// TIA Portal V20 export
FUNCTION_BLOCK "Sequence_1_SideTapeLoading"   // FB32854, LAD
TITLE = Sequence
// Sequence template programmend in ladder logic
// stored: IsIECCheckEnabled true, MemoryReserve 100, Namespace Unit1.Em4, SetENOAutomatically true
   VAR_INPUT
      unitStatus { ExternalAccessible := 'False'; ExternalVisible := 'False'; ExternalWritable := 'False'} : "LAF_typeUnitStatus";   // Current unit status o be used in this EM
   END_VAR
   VAR
      instSequenceLADControl { ExternalWritable := 'False'} : "LAF_ControlLadSequence";
      instSequenceLADStatus { ExternalWritable := 'False'} : "LAF_StatusLadSequence";
      statTonTime { ExternalWritable := 'False'} : Array[0..9999] of TON_TIME;
   END_VAR
   VAR_TEMP
      tempCustomerAction : Bool;   // Placeholder for possible actions
      tempDo_nothing_and_wait_for_init : Bool;   // Placeholder for doing nothing
      tempSafeStateCondition : Bool;   // Temp Condition for the equipment module to be in a safe state
   END_VAR
   VAR CONSTANT
      delayTime : Time := T#1000ms;
      STEP_IDLE : DInt := 1;
      JOB_1_STEP_1 : DInt := 101;
      JOB_1_STEP_10 : DInt := 110;
      JOB_1_STEP_20 : DInt := 120;
      JOB_1_STEP_30 : DInt := 130;
      JOB_1_STEP_40 : DInt := 140;
      JOB_1_STEP_50 : DInt := 150;
      JOB_1_STEP_90 : DInt := 190;
      JOB_2_STEP_1 : DInt := 201;
      JOB_2_STEP_10 : DInt := 210;
      JOB_2_STEP_20 : DInt := 220;
      JOB_2_STEP_30 : DInt := 230;
      JOB_2_STEP_40 : DInt := 240;
      JOB_2_STEP_50 : DInt := 250;
      JOB_2_STEP_60 : DInt := 260;
      JOB_2_STEP_90 : DInt := 290;
      JOB_3_STEP_10 : DInt := 310;
      JOB_3_STEP_20 : DInt := 320;
      JOB_3_STEP_30 : DInt := 330;
      JOB_3_STEP_40 : DInt := 340;
      STEP_IMMEDIATE_STOP : DInt := 9001;   // Step executed when an immediate stop command is triggered for the sequence (i.e. when unit is in state aborting)
      TO_DO_INSERT_ACTIONS_HERE : Bool := TRUE;   // Template : Add actions
      TO_DO_INSERT_CONDITION_FOR_TRANSITION_HERE : Bool := TRUE;   // Template : Add conditions
   END_VAR
   VAR_TEMP   // added for the SCL form of the ladder/FBD networks
      _w1 : Bool;
   END_VAR
BEGIN

REGION Network 1: BLOCK INFO HEADER
   // (company) / (C) Copyright (year)
   // ---------------------------------------------------------------------------------
   // Title:                             (Title of this block)
   // Comment/Function: (that is implemented in the block)
   // Library/Family:           (that the source is dedicated to)
   // Author:                        (department / person in charge / contact)
   // Target System:          (test system with FW version)
   // Engineering:              TIA Portal (SW version)
   // Restrictions:               (OB types, etc.)
   // Requirements:           (hardware, technological package, etc.)
   // ---------------------------------------------------------------------------------
   // Change log table:
   // Version          | Date             | Signature      | Expert in charge  | Changes applied ------------------------|----------------------|-------------------------|--------------------------------|-----------------------
   // 001.000.000 | yyyy-mm-dd | 0x00000000 | (name of expert) | First released version
END_REGION

REGION Network 2: DESCRIPTION
   // This is a template block provided by the Automation Framework. It can be used to create an own project.
   // The Block Info Header is prepared to put in your own data.
   // Description of the block could be added here and the docu created by Code2Docu.
END_REGION

REGION Network 3: *************** CONTROL **********************
END_REGION

REGION Network 4: Sequence Control ("Enter your Sequins number here")
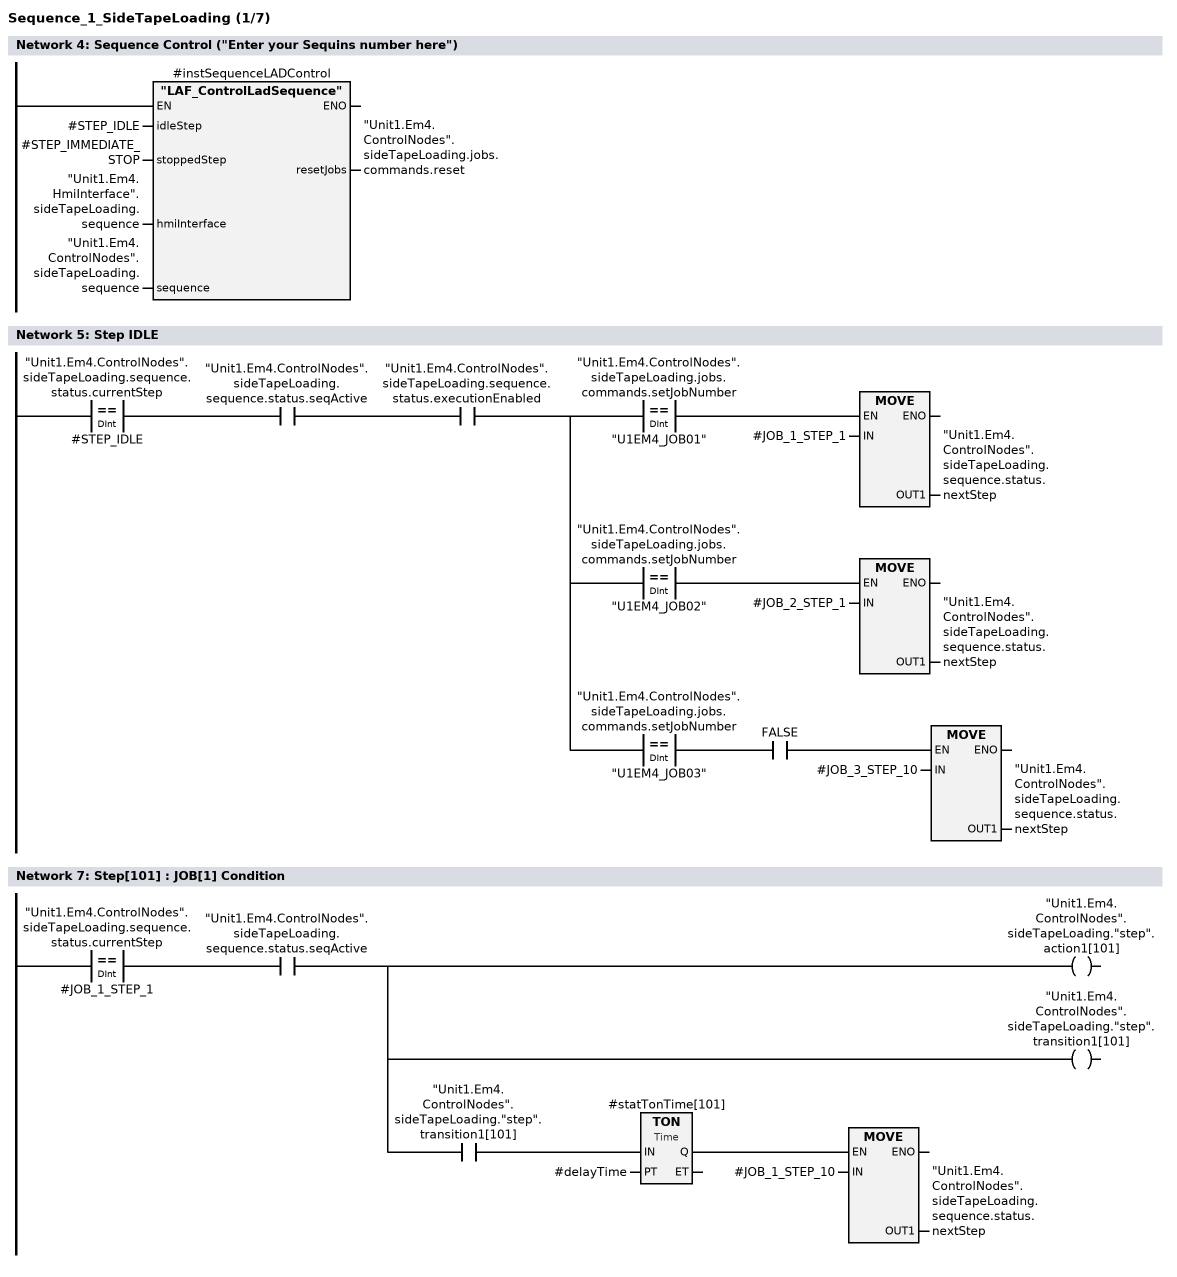
   RUNG wire#powerrail
      #instSequenceLADControl(idleStep := #STEP_IDLE, stoppedStep := #STEP_IMMEDIATE_STOP, hmiInterface := "Unit1.Em4.HmiInterface".sideTapeLoading.sequence, sequence := "Unit1.Em4.ControlNodes".sideTapeLoading.sequence, resetJobs => "Unit1.Em4.ControlNodes".sideTapeLoading.jobs.commands.reset)
   END_RUNG
   // the same network as SCL:
   #instSequenceLADControl(idleStep := #STEP_IDLE,   // "LAF_ControlLadSequence"
                           stoppedStep := #STEP_IMMEDIATE_STOP,
                           hmiInterface := "Unit1.Em4.HmiInterface".sideTapeLoading.sequence,
                           sequence := "Unit1.Em4.ControlNodes".sideTapeLoading.sequence,
                           resetJobs => "Unit1.Em4.ControlNodes".sideTapeLoading.jobs.commands.reset);
END_REGION

REGION Network 5: Step IDLE
   RUNG wire#powerrail
      { S7_Templates := "SrcType := DInt" } EQ_Contact(in1 := "Unit1.Em4.ControlNodes".sideTapeLoading.sequence.status.currentStep, in2 := #STEP_IDLE)
      Contact( "Unit1.Em4.ControlNodes".sideTapeLoading.sequence.status.seqActive )
      Contact( "Unit1.Em4.ControlNodes".sideTapeLoading.sequence.status.executionEnabled )
      wire#w1
      { S7_Templates := "SrcType := DInt" } EQ_Contact(in1 := "Unit1.Em4.ControlNodes".sideTapeLoading.jobs.commands.setJobNumber, in2 := "U1EM4_JOB01")
      Move(in := #JOB_1_STEP_1, out1 => "Unit1.Em4.ControlNodes".sideTapeLoading.sequence.status.nextStep)
   END_RUNG
   RUNG wire#w1
      { S7_Templates := "SrcType := DInt" } EQ_Contact(in1 := "Unit1.Em4.ControlNodes".sideTapeLoading.jobs.commands.setJobNumber, in2 := "U1EM4_JOB02")
      Move(in := #JOB_2_STEP_1, out1 => "Unit1.Em4.ControlNodes".sideTapeLoading.sequence.status.nextStep)
   END_RUNG
   RUNG wire#w1
      { S7_Templates := "SrcType := DInt" } EQ_Contact(in1 := "Unit1.Em4.ControlNodes".sideTapeLoading.jobs.commands.setJobNumber, in2 := "U1EM4_JOB03")
      Contact( FALSE )
      Move(in := #JOB_3_STEP_10, out1 => "Unit1.Em4.ControlNodes".sideTapeLoading.sequence.status.nextStep)
   END_RUNG
   // the same network as SCL:
   #_w1 := ("Unit1.Em4.ControlNodes".sideTapeLoading.sequence.status.currentStep = #STEP_IDLE) AND "Unit1.Em4.ControlNodes".sideTapeLoading.sequence.status.seqActive AND "Unit1.Em4.ControlNodes".sideTapeLoading.sequence.status.executionEnabled;
   IF #_w1 AND ("Unit1.Em4.ControlNodes".sideTapeLoading.jobs.commands.setJobNumber = "U1EM4_JOB01") THEN
       "Unit1.Em4.ControlNodes".sideTapeLoading.sequence.status.nextStep := #JOB_1_STEP_1;
   END_IF;
   IF #_w1 AND ("Unit1.Em4.ControlNodes".sideTapeLoading.jobs.commands.setJobNumber = "U1EM4_JOB02") THEN
       "Unit1.Em4.ControlNodes".sideTapeLoading.sequence.status.nextStep := #JOB_2_STEP_1;
   END_IF;
   IF #_w1 AND ("Unit1.Em4.ControlNodes".sideTapeLoading.jobs.commands.setJobNumber = "U1EM4_JOB03") AND FALSE THEN
       "Unit1.Em4.ControlNodes".sideTapeLoading.sequence.status.nextStep := #JOB_3_STEP_10;
   END_IF;
END_REGION

REGION Network 6: *************** JOB[1] HOMING *************************
END_REGION

REGION Network 7: Step[101] : JOB[1] Condition
   RUNG wire#powerrail
      { S7_Templates := "SrcType := DInt" } EQ_Contact(in1 := "Unit1.Em4.ControlNodes".sideTapeLoading.sequence.status.currentStep, in2 := #JOB_1_STEP_1)
      Contact( "Unit1.Em4.ControlNodes".sideTapeLoading.sequence.status.seqActive )
      wire#w1
      Coil( "Unit1.Em4.ControlNodes".sideTapeLoading."step".action1[101] )
   END_RUNG
   RUNG wire#w1
      Coil( "Unit1.Em4.ControlNodes".sideTapeLoading."step".transition1[101] )
   END_RUNG
   RUNG wire#w1
      Contact( "Unit1.Em4.ControlNodes".sideTapeLoading."step".transition1[101] )
      { S7_Templates := "time_type := Time" } #statTonTime[101].TON(pt := #delayTime, et =>)
      Move(in := #JOB_1_STEP_10, out1 => "Unit1.Em4.ControlNodes".sideTapeLoading.sequence.status.nextStep)
   END_RUNG
   // the same network as SCL:
   "Unit1.Em4.ControlNodes".sideTapeLoading."step".action1[101] := ("Unit1.Em4.ControlNodes".sideTapeLoading.sequence.status.currentStep = #JOB_1_STEP_1) AND "Unit1.Em4.ControlNodes".sideTapeLoading.sequence.status.seqActive;
   "Unit1.Em4.ControlNodes".sideTapeLoading."step".transition1[101] := ("Unit1.Em4.ControlNodes".sideTapeLoading.sequence.status.currentStep = #JOB_1_STEP_1) AND "Unit1.Em4.ControlNodes".sideTapeLoading.sequence.status.seqActive;
   #statTonTime[101].TON(IN := ("Unit1.Em4.ControlNodes".sideTapeLoading.sequence.status.currentStep = #JOB_1_STEP_1) AND "Unit1.Em4.ControlNodes".sideTapeLoading.sequence.status.seqActive AND "Unit1.Em4.ControlNodes".sideTapeLoading."step".transition1[101],
                         PT := #delayTime);
   IF #statTonTime[101].Q THEN
       "Unit1.Em4.ControlNodes".sideTapeLoading.sequence.status.nextStep := #JOB_1_STEP_10;
   END_IF;
END_REGION

REGION Network 8: Step[110] : Side Tape Loading Down
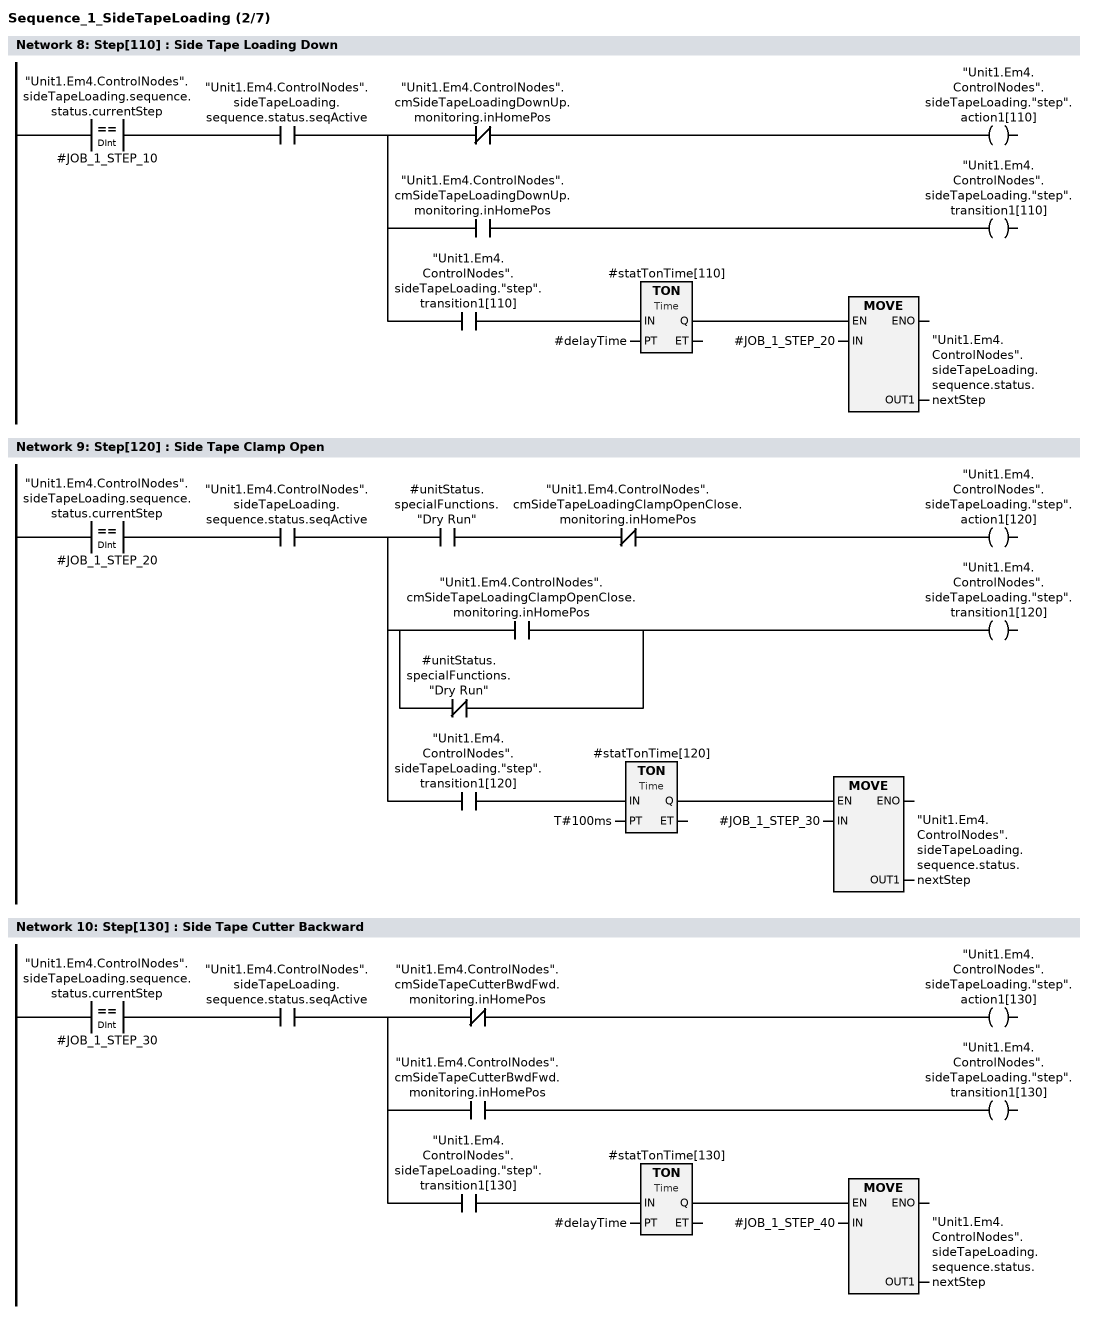
   RUNG wire#powerrail
      { S7_Templates := "SrcType := DInt" } EQ_Contact(in1 := "Unit1.Em4.ControlNodes".sideTapeLoading.sequence.status.currentStep, in2 := #JOB_1_STEP_10)
      Contact( "Unit1.Em4.ControlNodes".sideTapeLoading.sequence.status.seqActive )
      wire#w1
      I_Contact( "Unit1.Em4.ControlNodes".cmSideTapeLoadingDownUp.monitoring.inHomePos )
      Coil( "Unit1.Em4.ControlNodes".sideTapeLoading."step".action1[110] )
   END_RUNG
   RUNG wire#w1
      Contact( "Unit1.Em4.ControlNodes".cmSideTapeLoadingDownUp.monitoring.inHomePos )
      Coil( "Unit1.Em4.ControlNodes".sideTapeLoading."step".transition1[110] )
   END_RUNG
   RUNG wire#w1
      Contact( "Unit1.Em4.ControlNodes".sideTapeLoading."step".transition1[110] )
      { S7_Templates := "time_type := Time" } #statTonTime[110].TON(pt := #delayTime, et =>)
      Move(in := #JOB_1_STEP_20, out1 => "Unit1.Em4.ControlNodes".sideTapeLoading.sequence.status.nextStep)
   END_RUNG
   // the same network as SCL:
   #_w1 := ("Unit1.Em4.ControlNodes".sideTapeLoading.sequence.status.currentStep = #JOB_1_STEP_10) AND "Unit1.Em4.ControlNodes".sideTapeLoading.sequence.status.seqActive;
   "Unit1.Em4.ControlNodes".sideTapeLoading."step".action1[110] := #_w1 AND NOT "Unit1.Em4.ControlNodes".cmSideTapeLoadingDownUp.monitoring.inHomePos;
   "Unit1.Em4.ControlNodes".sideTapeLoading."step".transition1[110] := #_w1 AND "Unit1.Em4.ControlNodes".cmSideTapeLoadingDownUp.monitoring.inHomePos;
   #statTonTime[110].TON(IN := #_w1 AND "Unit1.Em4.ControlNodes".sideTapeLoading."step".transition1[110],
                         PT := #delayTime);
   IF #statTonTime[110].Q THEN
       "Unit1.Em4.ControlNodes".sideTapeLoading.sequence.status.nextStep := #JOB_1_STEP_20;
   END_IF;
END_REGION

REGION Network 9: Step[120] : Side Tape Clamp Open
   RUNG wire#powerrail
      { S7_Templates := "SrcType := DInt" } EQ_Contact(in1 := "Unit1.Em4.ControlNodes".sideTapeLoading.sequence.status.currentStep, in2 := #JOB_1_STEP_20)
      Contact( "Unit1.Em4.ControlNodes".sideTapeLoading.sequence.status.seqActive )
      wire#w1
      Contact( #unitStatus.specialFunctions."Dry Run" )
      I_Contact( "Unit1.Em4.ControlNodes".cmSideTapeLoadingClampOpenClose.monitoring.inHomePos )
      Coil( "Unit1.Em4.ControlNodes".sideTapeLoading."step".action1[120] )
   END_RUNG
   RUNG wire#w1
      Contact( "Unit1.Em4.ControlNodes".cmSideTapeLoadingClampOpenClose.monitoring.inHomePos )
      wire#w2
      Coil( "Unit1.Em4.ControlNodes".sideTapeLoading."step".transition1[120] )
   END_RUNG
   RUNG wire#w1
      I_Contact( #unitStatus.specialFunctions."Dry Run" )
   END_RUNG wire#w2
   RUNG wire#w1
      Contact( "Unit1.Em4.ControlNodes".sideTapeLoading."step".transition1[120] )
      { S7_Templates := "time_type := Time" } #statTonTime[120].TON(pt := T#100ms, et =>)
      Move(in := #JOB_1_STEP_30, out1 => "Unit1.Em4.ControlNodes".sideTapeLoading.sequence.status.nextStep)
   END_RUNG
   // the same network as SCL:
   #_w1 := ("Unit1.Em4.ControlNodes".sideTapeLoading.sequence.status.currentStep = #JOB_1_STEP_20) AND "Unit1.Em4.ControlNodes".sideTapeLoading.sequence.status.seqActive;
   "Unit1.Em4.ControlNodes".sideTapeLoading."step".action1[120] := #_w1 AND #unitStatus.specialFunctions."Dry Run" AND NOT "Unit1.Em4.ControlNodes".cmSideTapeLoadingClampOpenClose.monitoring.inHomePos;
   "Unit1.Em4.ControlNodes".sideTapeLoading."step".transition1[120] := #_w1 AND ("Unit1.Em4.ControlNodes".cmSideTapeLoadingClampOpenClose.monitoring.inHomePos OR NOT #unitStatus.specialFunctions."Dry Run");
   #statTonTime[120].TON(IN := #_w1 AND "Unit1.Em4.ControlNodes".sideTapeLoading."step".transition1[120],
                         PT := T#100ms);
   IF #statTonTime[120].Q THEN
       "Unit1.Em4.ControlNodes".sideTapeLoading.sequence.status.nextStep := #JOB_1_STEP_30;
   END_IF;
END_REGION

REGION Network 10: Step[130] : Side Tape Cutter Backward
   RUNG wire#powerrail
      { S7_Templates := "SrcType := DInt" } EQ_Contact(in1 := "Unit1.Em4.ControlNodes".sideTapeLoading.sequence.status.currentStep, in2 := #JOB_1_STEP_30)
      Contact( "Unit1.Em4.ControlNodes".sideTapeLoading.sequence.status.seqActive )
      wire#w1
      I_Contact( "Unit1.Em4.ControlNodes".cmSideTapeCutterBwdFwd.monitoring.inHomePos )
      Coil( "Unit1.Em4.ControlNodes".sideTapeLoading."step".action1[130] )
   END_RUNG
   RUNG wire#w1
      Contact( "Unit1.Em4.ControlNodes".cmSideTapeCutterBwdFwd.monitoring.inHomePos )
      Coil( "Unit1.Em4.ControlNodes".sideTapeLoading."step".transition1[130] )
   END_RUNG
   RUNG wire#w1
      Contact( "Unit1.Em4.ControlNodes".sideTapeLoading."step".transition1[130] )
      { S7_Templates := "time_type := Time" } #statTonTime[130].TON(pt := #delayTime, et =>)
      Move(in := #JOB_1_STEP_40, out1 => "Unit1.Em4.ControlNodes".sideTapeLoading.sequence.status.nextStep)
   END_RUNG
   // the same network as SCL:
   #_w1 := ("Unit1.Em4.ControlNodes".sideTapeLoading.sequence.status.currentStep = #JOB_1_STEP_30) AND "Unit1.Em4.ControlNodes".sideTapeLoading.sequence.status.seqActive;
   "Unit1.Em4.ControlNodes".sideTapeLoading."step".action1[130] := #_w1 AND NOT "Unit1.Em4.ControlNodes".cmSideTapeCutterBwdFwd.monitoring.inHomePos;
   "Unit1.Em4.ControlNodes".sideTapeLoading."step".transition1[130] := #_w1 AND "Unit1.Em4.ControlNodes".cmSideTapeCutterBwdFwd.monitoring.inHomePos;
   #statTonTime[130].TON(IN := #_w1 AND "Unit1.Em4.ControlNodes".sideTapeLoading."step".transition1[130],
                         PT := #delayTime);
   IF #statTonTime[130].Q THEN
       "Unit1.Em4.ControlNodes".sideTapeLoading.sequence.status.nextStep := #JOB_1_STEP_40;
   END_IF;
END_REGION

REGION Network 11: Step[140] : Side Tape Cutter Clamp Forward
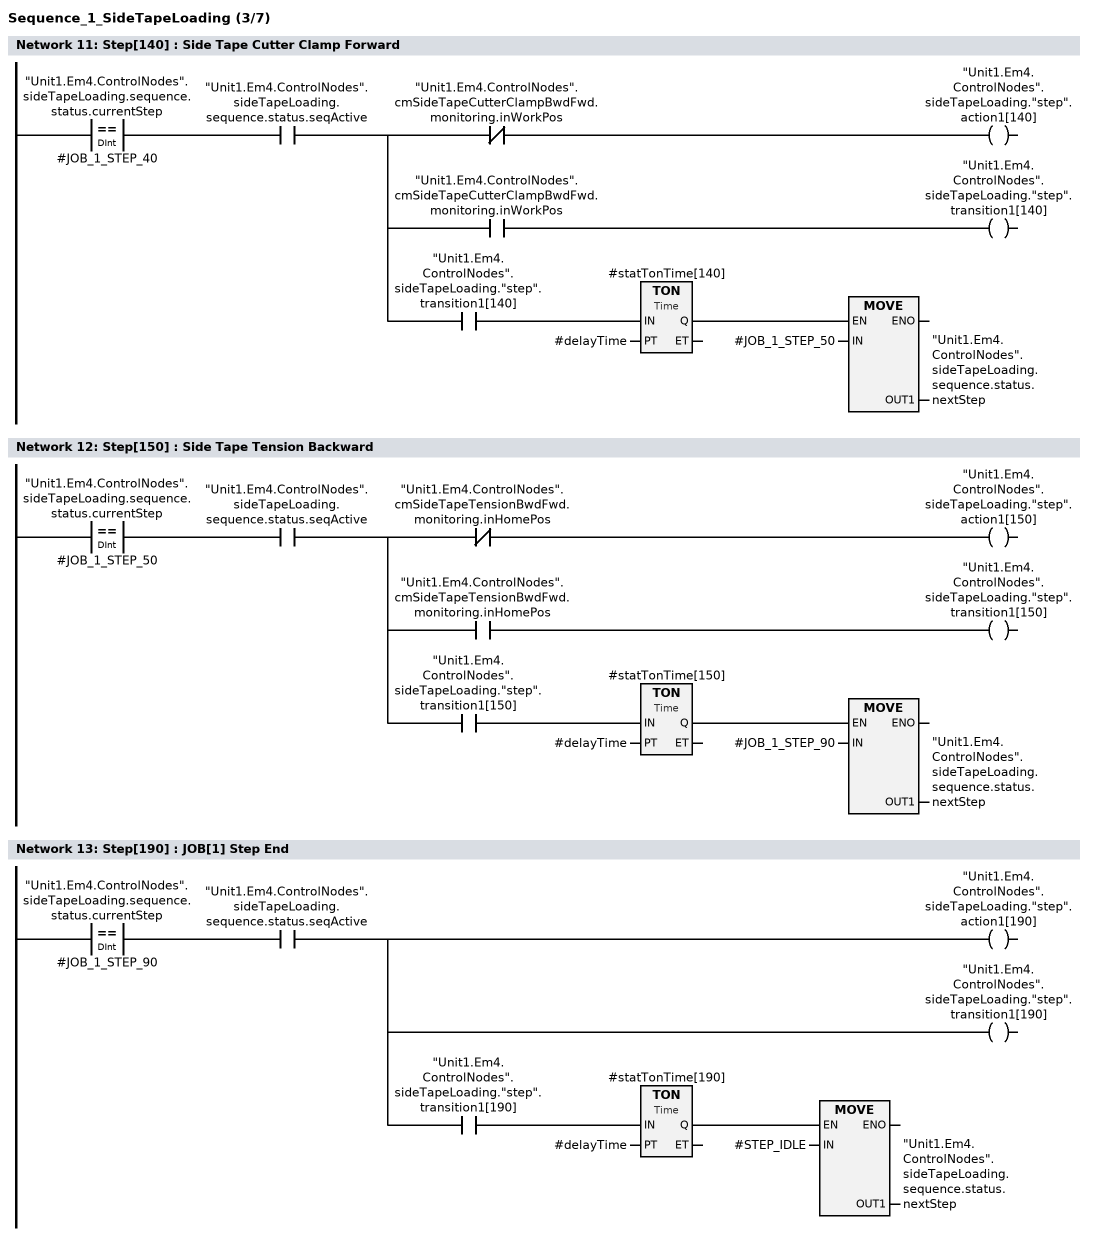
   RUNG wire#powerrail
      { S7_Templates := "SrcType := DInt" } EQ_Contact(in1 := "Unit1.Em4.ControlNodes".sideTapeLoading.sequence.status.currentStep, in2 := #JOB_1_STEP_40)
      Contact( "Unit1.Em4.ControlNodes".sideTapeLoading.sequence.status.seqActive )
      wire#w1
      I_Contact( "Unit1.Em4.ControlNodes".cmSideTapeCutterClampBwdFwd.monitoring.inWorkPos )
      Coil( "Unit1.Em4.ControlNodes".sideTapeLoading."step".action1[140] )
   END_RUNG
   RUNG wire#w1
      Contact( "Unit1.Em4.ControlNodes".cmSideTapeCutterClampBwdFwd.monitoring.inWorkPos )
      Coil( "Unit1.Em4.ControlNodes".sideTapeLoading."step".transition1[140] )
   END_RUNG
   RUNG wire#w1
      Contact( "Unit1.Em4.ControlNodes".sideTapeLoading."step".transition1[140] )
      { S7_Templates := "time_type := Time" } #statTonTime[140].TON(pt := #delayTime, et =>)
      Move(in := #JOB_1_STEP_50, out1 => "Unit1.Em4.ControlNodes".sideTapeLoading.sequence.status.nextStep)
   END_RUNG
   // the same network as SCL:
   #_w1 := ("Unit1.Em4.ControlNodes".sideTapeLoading.sequence.status.currentStep = #JOB_1_STEP_40) AND "Unit1.Em4.ControlNodes".sideTapeLoading.sequence.status.seqActive;
   "Unit1.Em4.ControlNodes".sideTapeLoading."step".action1[140] := #_w1 AND NOT "Unit1.Em4.ControlNodes".cmSideTapeCutterClampBwdFwd.monitoring.inWorkPos;
   "Unit1.Em4.ControlNodes".sideTapeLoading."step".transition1[140] := #_w1 AND "Unit1.Em4.ControlNodes".cmSideTapeCutterClampBwdFwd.monitoring.inWorkPos;
   #statTonTime[140].TON(IN := #_w1 AND "Unit1.Em4.ControlNodes".sideTapeLoading."step".transition1[140],
                         PT := #delayTime);
   IF #statTonTime[140].Q THEN
       "Unit1.Em4.ControlNodes".sideTapeLoading.sequence.status.nextStep := #JOB_1_STEP_50;
   END_IF;
END_REGION

REGION Network 12: Step[150] : Side Tape Tension Backward
   RUNG wire#powerrail
      { S7_Templates := "SrcType := DInt" } EQ_Contact(in1 := "Unit1.Em4.ControlNodes".sideTapeLoading.sequence.status.currentStep, in2 := #JOB_1_STEP_50)
      Contact( "Unit1.Em4.ControlNodes".sideTapeLoading.sequence.status.seqActive )
      wire#w1
      I_Contact( "Unit1.Em4.ControlNodes".cmSideTapeTensionBwdFwd.monitoring.inHomePos )
      Coil( "Unit1.Em4.ControlNodes".sideTapeLoading."step".action1[150] )
   END_RUNG
   RUNG wire#w1
      Contact( "Unit1.Em4.ControlNodes".cmSideTapeTensionBwdFwd.monitoring.inHomePos )
      Coil( "Unit1.Em4.ControlNodes".sideTapeLoading."step".transition1[150] )
   END_RUNG
   RUNG wire#w1
      Contact( "Unit1.Em4.ControlNodes".sideTapeLoading."step".transition1[150] )
      { S7_Templates := "time_type := Time" } #statTonTime[150].TON(pt := #delayTime, et =>)
      Move(in := #JOB_1_STEP_90, out1 => "Unit1.Em4.ControlNodes".sideTapeLoading.sequence.status.nextStep)
   END_RUNG
   // the same network as SCL:
   #_w1 := ("Unit1.Em4.ControlNodes".sideTapeLoading.sequence.status.currentStep = #JOB_1_STEP_50) AND "Unit1.Em4.ControlNodes".sideTapeLoading.sequence.status.seqActive;
   "Unit1.Em4.ControlNodes".sideTapeLoading."step".action1[150] := #_w1 AND NOT "Unit1.Em4.ControlNodes".cmSideTapeTensionBwdFwd.monitoring.inHomePos;
   "Unit1.Em4.ControlNodes".sideTapeLoading."step".transition1[150] := #_w1 AND "Unit1.Em4.ControlNodes".cmSideTapeTensionBwdFwd.monitoring.inHomePos;
   #statTonTime[150].TON(IN := #_w1 AND "Unit1.Em4.ControlNodes".sideTapeLoading."step".transition1[150],
                         PT := #delayTime);
   IF #statTonTime[150].Q THEN
       "Unit1.Em4.ControlNodes".sideTapeLoading.sequence.status.nextStep := #JOB_1_STEP_90;
   END_IF;
END_REGION

REGION Network 13: Step[190] : JOB[1] Step End
   RUNG wire#powerrail
      { S7_Templates := "SrcType := DInt" } EQ_Contact(in1 := "Unit1.Em4.ControlNodes".sideTapeLoading.sequence.status.currentStep, in2 := #JOB_1_STEP_90)
      Contact( "Unit1.Em4.ControlNodes".sideTapeLoading.sequence.status.seqActive )
      wire#w1
      Coil( "Unit1.Em4.ControlNodes".sideTapeLoading."step".action1[190] )
   END_RUNG
   RUNG wire#w1
      Coil( "Unit1.Em4.ControlNodes".sideTapeLoading."step".transition1[190] )
   END_RUNG
   RUNG wire#w1
      Contact( "Unit1.Em4.ControlNodes".sideTapeLoading."step".transition1[190] )
      { S7_Templates := "time_type := Time" } #statTonTime[190].TON(pt := #delayTime, et =>)
      Move(in := #STEP_IDLE, out1 => "Unit1.Em4.ControlNodes".sideTapeLoading.sequence.status.nextStep)
   END_RUNG
   // the same network as SCL:
   "Unit1.Em4.ControlNodes".sideTapeLoading."step".action1[190] := ("Unit1.Em4.ControlNodes".sideTapeLoading.sequence.status.currentStep = #JOB_1_STEP_90) AND "Unit1.Em4.ControlNodes".sideTapeLoading.sequence.status.seqActive;
   "Unit1.Em4.ControlNodes".sideTapeLoading."step".transition1[190] := ("Unit1.Em4.ControlNodes".sideTapeLoading.sequence.status.currentStep = #JOB_1_STEP_90) AND "Unit1.Em4.ControlNodes".sideTapeLoading.sequence.status.seqActive;
   #statTonTime[190].TON(IN := ("Unit1.Em4.ControlNodes".sideTapeLoading.sequence.status.currentStep = #JOB_1_STEP_90) AND "Unit1.Em4.ControlNodes".sideTapeLoading.sequence.status.seqActive AND "Unit1.Em4.ControlNodes".sideTapeLoading."step".transition1[190],
                         PT := #delayTime);
   IF #statTonTime[190].Q THEN
       "Unit1.Em4.ControlNodes".sideTapeLoading.sequence.status.nextStep := #STEP_IDLE;
   END_IF;
END_REGION

REGION Network 14: *************** JOB[2] SIDE TAPE CHARGE=AUTO *************************
END_REGION

REGION Network 15: Step[201] : JOB[2] Condition
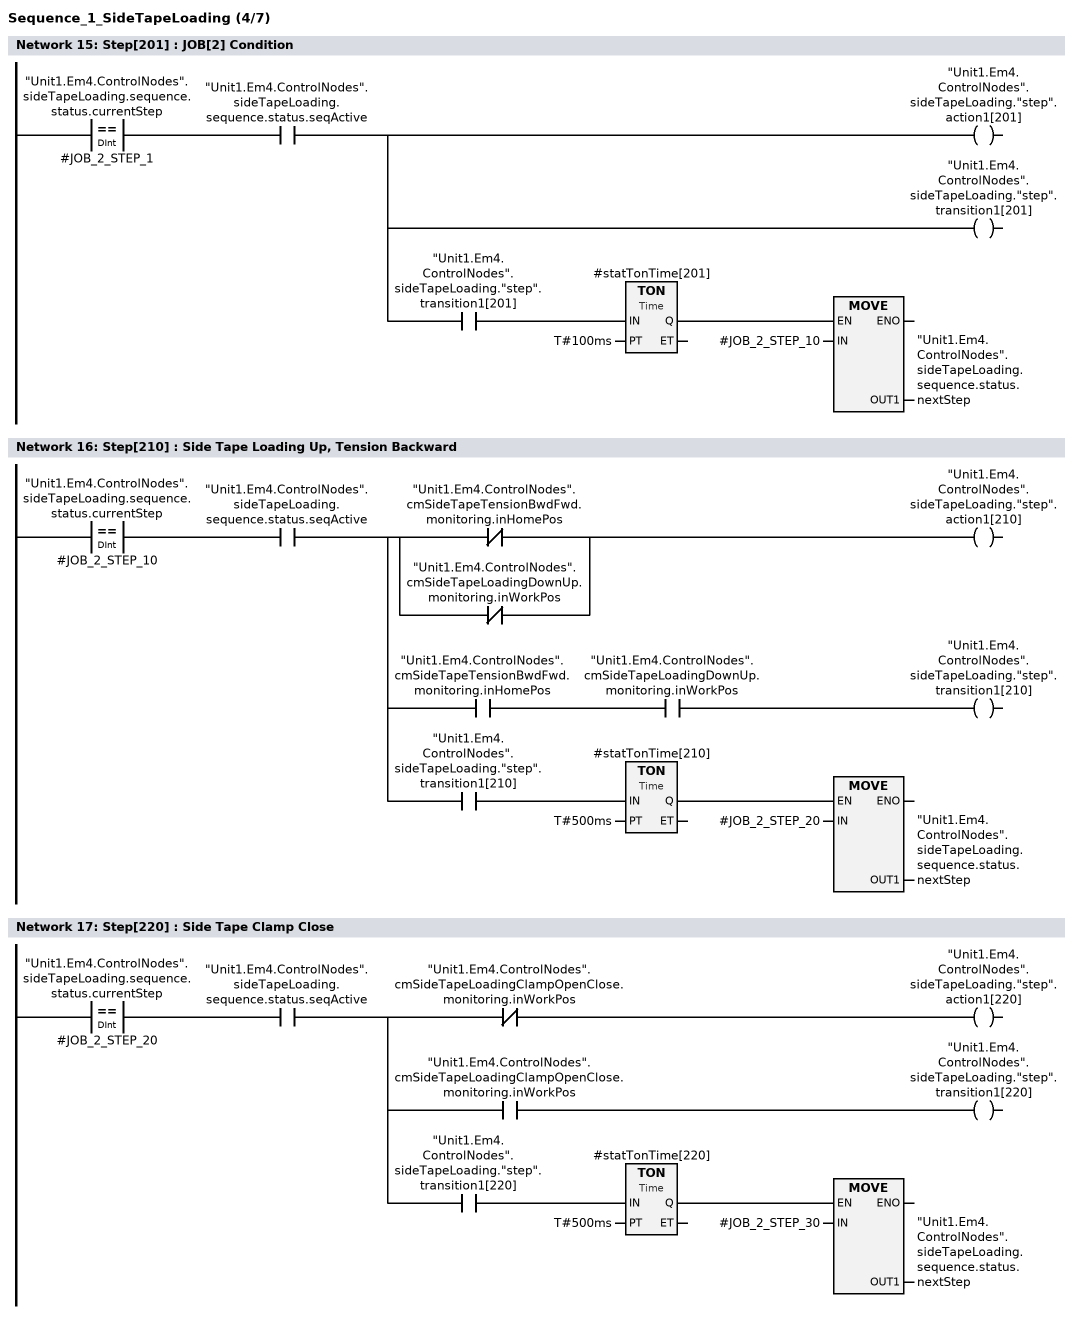
   RUNG wire#powerrail
      { S7_Templates := "SrcType := DInt" } EQ_Contact(in1 := "Unit1.Em4.ControlNodes".sideTapeLoading.sequence.status.currentStep, in2 := #JOB_2_STEP_1)
      Contact( "Unit1.Em4.ControlNodes".sideTapeLoading.sequence.status.seqActive )
      wire#w1
      Coil( "Unit1.Em4.ControlNodes".sideTapeLoading."step".action1[201] )
   END_RUNG
   RUNG wire#w1
      Coil( "Unit1.Em4.ControlNodes".sideTapeLoading."step".transition1[201] )
   END_RUNG
   RUNG wire#w1
      Contact( "Unit1.Em4.ControlNodes".sideTapeLoading."step".transition1[201] )
      { S7_Templates := "time_type := Time" } #statTonTime[201].TON(pt := T#100ms, et =>)
      Move(in := #JOB_2_STEP_10, out1 => "Unit1.Em4.ControlNodes".sideTapeLoading.sequence.status.nextStep)
   END_RUNG
   // the same network as SCL:
   "Unit1.Em4.ControlNodes".sideTapeLoading."step".action1[201] := ("Unit1.Em4.ControlNodes".sideTapeLoading.sequence.status.currentStep = #JOB_2_STEP_1) AND "Unit1.Em4.ControlNodes".sideTapeLoading.sequence.status.seqActive;
   "Unit1.Em4.ControlNodes".sideTapeLoading."step".transition1[201] := ("Unit1.Em4.ControlNodes".sideTapeLoading.sequence.status.currentStep = #JOB_2_STEP_1) AND "Unit1.Em4.ControlNodes".sideTapeLoading.sequence.status.seqActive;
   #statTonTime[201].TON(IN := ("Unit1.Em4.ControlNodes".sideTapeLoading.sequence.status.currentStep = #JOB_2_STEP_1) AND "Unit1.Em4.ControlNodes".sideTapeLoading.sequence.status.seqActive AND "Unit1.Em4.ControlNodes".sideTapeLoading."step".transition1[201],
                         PT := T#100ms);
   IF #statTonTime[201].Q THEN
       "Unit1.Em4.ControlNodes".sideTapeLoading.sequence.status.nextStep := #JOB_2_STEP_10;
   END_IF;
END_REGION

REGION Network 16: Step[210] : Side Tape Loading Up, Tension Backward
   RUNG wire#powerrail
      { S7_Templates := "SrcType := DInt" } EQ_Contact(in1 := "Unit1.Em4.ControlNodes".sideTapeLoading.sequence.status.currentStep, in2 := #JOB_2_STEP_10)
      Contact( "Unit1.Em4.ControlNodes".sideTapeLoading.sequence.status.seqActive )
      wire#w1
      I_Contact( "Unit1.Em4.ControlNodes".cmSideTapeTensionBwdFwd.monitoring.inHomePos )
      wire#w2
      Coil( "Unit1.Em4.ControlNodes".sideTapeLoading."step".action1[210] )
   END_RUNG
   RUNG wire#w1
      I_Contact( "Unit1.Em4.ControlNodes".cmSideTapeLoadingDownUp.monitoring.inWorkPos )
   END_RUNG wire#w2
   RUNG wire#w1
      Contact( "Unit1.Em4.ControlNodes".cmSideTapeTensionBwdFwd.monitoring.inHomePos )
      Contact( "Unit1.Em4.ControlNodes".cmSideTapeLoadingDownUp.monitoring.inWorkPos )
      Coil( "Unit1.Em4.ControlNodes".sideTapeLoading."step".transition1[210] )
   END_RUNG
   RUNG wire#w1
      Contact( "Unit1.Em4.ControlNodes".sideTapeLoading."step".transition1[210] )
      { S7_Templates := "time_type := Time" } #statTonTime[210].TON(pt := T#500ms, et =>)
      Move(in := #JOB_2_STEP_20, out1 => "Unit1.Em4.ControlNodes".sideTapeLoading.sequence.status.nextStep)
   END_RUNG
   // the same network as SCL:
   #_w1 := ("Unit1.Em4.ControlNodes".sideTapeLoading.sequence.status.currentStep = #JOB_2_STEP_10) AND "Unit1.Em4.ControlNodes".sideTapeLoading.sequence.status.seqActive;
   "Unit1.Em4.ControlNodes".sideTapeLoading."step".action1[210] := #_w1 AND (NOT "Unit1.Em4.ControlNodes".cmSideTapeTensionBwdFwd.monitoring.inHomePos OR NOT "Unit1.Em4.ControlNodes".cmSideTapeLoadingDownUp.monitoring.inWorkPos);
   "Unit1.Em4.ControlNodes".sideTapeLoading."step".transition1[210] := #_w1 AND "Unit1.Em4.ControlNodes".cmSideTapeTensionBwdFwd.monitoring.inHomePos AND "Unit1.Em4.ControlNodes".cmSideTapeLoadingDownUp.monitoring.inWorkPos;
   #statTonTime[210].TON(IN := #_w1 AND "Unit1.Em4.ControlNodes".sideTapeLoading."step".transition1[210],
                         PT := T#500ms);
   IF #statTonTime[210].Q THEN
       "Unit1.Em4.ControlNodes".sideTapeLoading.sequence.status.nextStep := #JOB_2_STEP_20;
   END_IF;
END_REGION

REGION Network 17: Step[220] : Side Tape Clamp Close
   RUNG wire#powerrail
      { S7_Templates := "SrcType := DInt" } EQ_Contact(in1 := "Unit1.Em4.ControlNodes".sideTapeLoading.sequence.status.currentStep, in2 := #JOB_2_STEP_20)
      Contact( "Unit1.Em4.ControlNodes".sideTapeLoading.sequence.status.seqActive )
      wire#w1
      I_Contact( "Unit1.Em4.ControlNodes".cmSideTapeLoadingClampOpenClose.monitoring.inWorkPos )
      Coil( "Unit1.Em4.ControlNodes".sideTapeLoading."step".action1[220] )
   END_RUNG
   RUNG wire#w1
      Contact( "Unit1.Em4.ControlNodes".cmSideTapeLoadingClampOpenClose.monitoring.inWorkPos )
      Coil( "Unit1.Em4.ControlNodes".sideTapeLoading."step".transition1[220] )
   END_RUNG
   RUNG wire#w1
      Contact( "Unit1.Em4.ControlNodes".sideTapeLoading."step".transition1[220] )
      { S7_Templates := "time_type := Time" } #statTonTime[220].TON(pt := T#500ms, et =>)
      Move(in := #JOB_2_STEP_30, out1 => "Unit1.Em4.ControlNodes".sideTapeLoading.sequence.status.nextStep)
   END_RUNG
   // the same network as SCL:
   #_w1 := ("Unit1.Em4.ControlNodes".sideTapeLoading.sequence.status.currentStep = #JOB_2_STEP_20) AND "Unit1.Em4.ControlNodes".sideTapeLoading.sequence.status.seqActive;
   "Unit1.Em4.ControlNodes".sideTapeLoading."step".action1[220] := #_w1 AND NOT "Unit1.Em4.ControlNodes".cmSideTapeLoadingClampOpenClose.monitoring.inWorkPos;
   "Unit1.Em4.ControlNodes".sideTapeLoading."step".transition1[220] := #_w1 AND "Unit1.Em4.ControlNodes".cmSideTapeLoadingClampOpenClose.monitoring.inWorkPos;
   #statTonTime[220].TON(IN := #_w1 AND "Unit1.Em4.ControlNodes".sideTapeLoading."step".transition1[220],
                         PT := T#500ms);
   IF #statTonTime[220].Q THEN
       "Unit1.Em4.ControlNodes".sideTapeLoading.sequence.status.nextStep := #JOB_2_STEP_30;
   END_IF;
END_REGION

REGION Network 18: Step[230] : Side Tape Cutter Clamp Backward
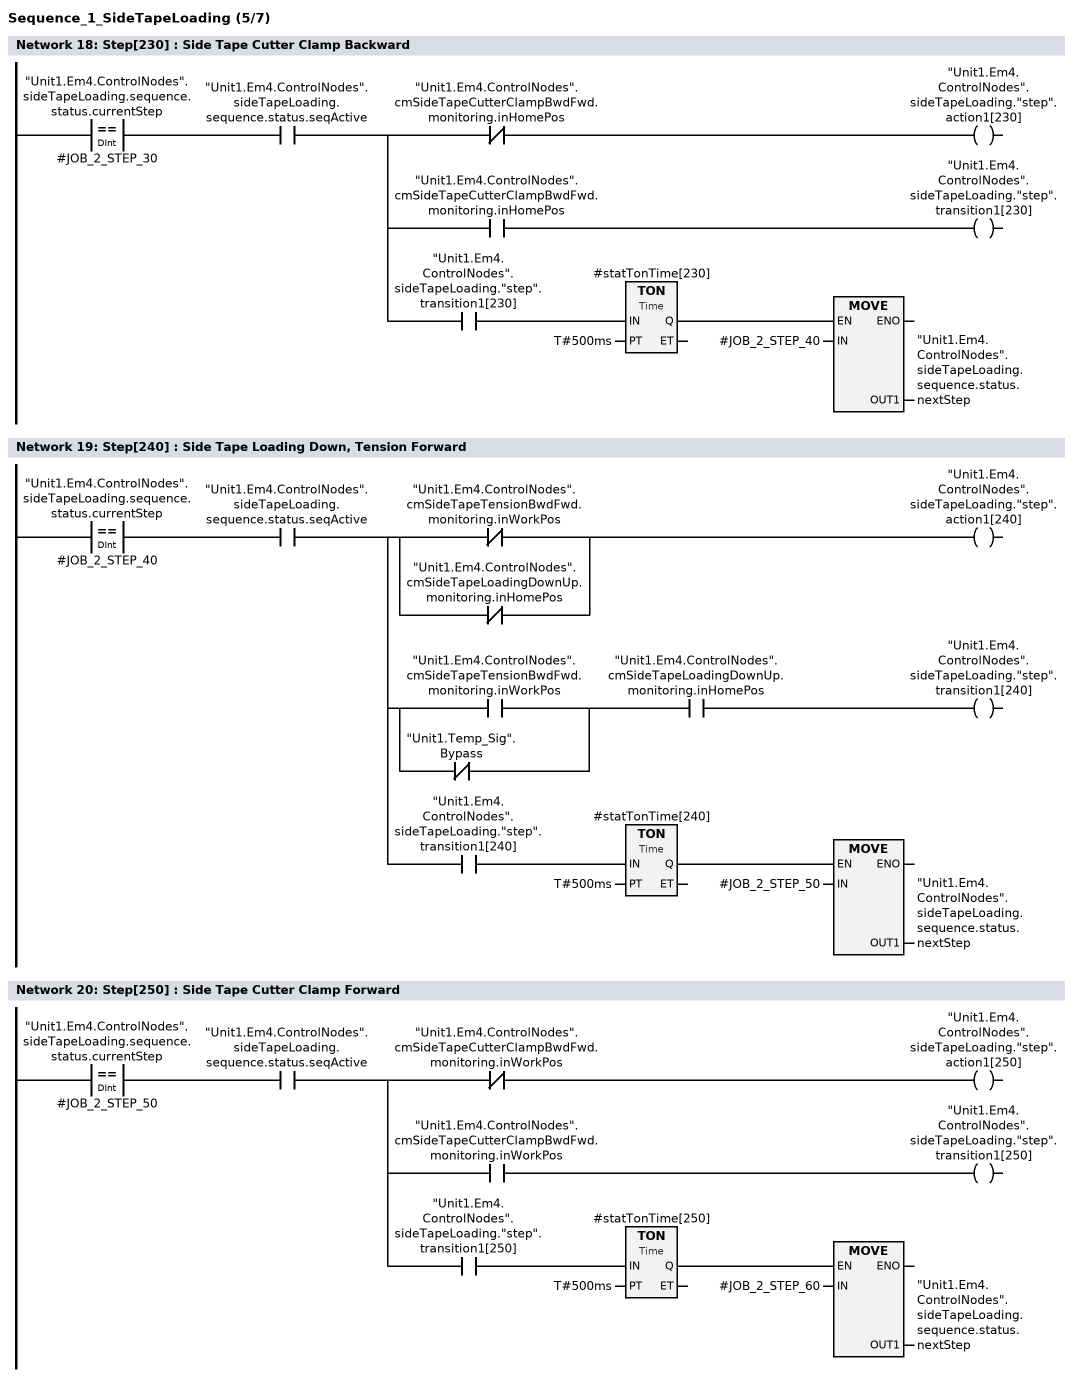
   RUNG wire#powerrail
      { S7_Templates := "SrcType := DInt" } EQ_Contact(in1 := "Unit1.Em4.ControlNodes".sideTapeLoading.sequence.status.currentStep, in2 := #JOB_2_STEP_30)
      Contact( "Unit1.Em4.ControlNodes".sideTapeLoading.sequence.status.seqActive )
      wire#w1
      I_Contact( "Unit1.Em4.ControlNodes".cmSideTapeCutterClampBwdFwd.monitoring.inHomePos )
      Coil( "Unit1.Em4.ControlNodes".sideTapeLoading."step".action1[230] )
   END_RUNG
   RUNG wire#w1
      Contact( "Unit1.Em4.ControlNodes".cmSideTapeCutterClampBwdFwd.monitoring.inHomePos )
      Coil( "Unit1.Em4.ControlNodes".sideTapeLoading."step".transition1[230] )
   END_RUNG
   RUNG wire#w1
      Contact( "Unit1.Em4.ControlNodes".sideTapeLoading."step".transition1[230] )
      { S7_Templates := "time_type := Time" } #statTonTime[230].TON(pt := T#500ms, et =>)
      Move(in := #JOB_2_STEP_40, out1 => "Unit1.Em4.ControlNodes".sideTapeLoading.sequence.status.nextStep)
   END_RUNG
   // the same network as SCL:
   #_w1 := ("Unit1.Em4.ControlNodes".sideTapeLoading.sequence.status.currentStep = #JOB_2_STEP_30) AND "Unit1.Em4.ControlNodes".sideTapeLoading.sequence.status.seqActive;
   "Unit1.Em4.ControlNodes".sideTapeLoading."step".action1[230] := #_w1 AND NOT "Unit1.Em4.ControlNodes".cmSideTapeCutterClampBwdFwd.monitoring.inHomePos;
   "Unit1.Em4.ControlNodes".sideTapeLoading."step".transition1[230] := #_w1 AND "Unit1.Em4.ControlNodes".cmSideTapeCutterClampBwdFwd.monitoring.inHomePos;
   #statTonTime[230].TON(IN := #_w1 AND "Unit1.Em4.ControlNodes".sideTapeLoading."step".transition1[230],
                         PT := T#500ms);
   IF #statTonTime[230].Q THEN
       "Unit1.Em4.ControlNodes".sideTapeLoading.sequence.status.nextStep := #JOB_2_STEP_40;
   END_IF;
END_REGION

REGION Network 19: Step[240] : Side Tape Loading Down, Tension Forward
   RUNG wire#powerrail
      { S7_Templates := "SrcType := DInt" } EQ_Contact(in1 := "Unit1.Em4.ControlNodes".sideTapeLoading.sequence.status.currentStep, in2 := #JOB_2_STEP_40)
      Contact( "Unit1.Em4.ControlNodes".sideTapeLoading.sequence.status.seqActive )
      wire#w1
      I_Contact( "Unit1.Em4.ControlNodes".cmSideTapeTensionBwdFwd.monitoring.inWorkPos )
      wire#w2
      Coil( "Unit1.Em4.ControlNodes".sideTapeLoading."step".action1[240] )
   END_RUNG
   RUNG wire#w1
      I_Contact( "Unit1.Em4.ControlNodes".cmSideTapeLoadingDownUp.monitoring.inHomePos )
   END_RUNG wire#w2
   RUNG wire#w1
      Contact( "Unit1.Em4.ControlNodes".cmSideTapeTensionBwdFwd.monitoring.inWorkPos )
      wire#w3
      Contact( "Unit1.Em4.ControlNodes".cmSideTapeLoadingDownUp.monitoring.inHomePos )
      Coil( "Unit1.Em4.ControlNodes".sideTapeLoading."step".transition1[240] )
   END_RUNG
   RUNG wire#w1
      I_Contact( "Unit1.Temp_Sig".Bypass )
   END_RUNG wire#w3
   RUNG wire#w1
      Contact( "Unit1.Em4.ControlNodes".sideTapeLoading."step".transition1[240] )
      { S7_Templates := "time_type := Time" } #statTonTime[240].TON(pt := T#500ms, et =>)
      Move(in := #JOB_2_STEP_50, out1 => "Unit1.Em4.ControlNodes".sideTapeLoading.sequence.status.nextStep)
   END_RUNG
   // the same network as SCL:
   #_w1 := ("Unit1.Em4.ControlNodes".sideTapeLoading.sequence.status.currentStep = #JOB_2_STEP_40) AND "Unit1.Em4.ControlNodes".sideTapeLoading.sequence.status.seqActive;
   "Unit1.Em4.ControlNodes".sideTapeLoading."step".action1[240] := #_w1 AND (NOT "Unit1.Em4.ControlNodes".cmSideTapeTensionBwdFwd.monitoring.inWorkPos OR NOT "Unit1.Em4.ControlNodes".cmSideTapeLoadingDownUp.monitoring.inHomePos);
   "Unit1.Em4.ControlNodes".sideTapeLoading."step".transition1[240] := #_w1 AND ("Unit1.Em4.ControlNodes".cmSideTapeTensionBwdFwd.monitoring.inWorkPos OR NOT "Unit1.Temp_Sig".Bypass) AND "Unit1.Em4.ControlNodes".cmSideTapeLoadingDownUp.monitoring.inHomePos;
   #statTonTime[240].TON(IN := #_w1 AND "Unit1.Em4.ControlNodes".sideTapeLoading."step".transition1[240],
                         PT := T#500ms);
   IF #statTonTime[240].Q THEN
       "Unit1.Em4.ControlNodes".sideTapeLoading.sequence.status.nextStep := #JOB_2_STEP_50;
   END_IF;
END_REGION

REGION Network 20: Step[250] : Side Tape Cutter Clamp Forward
   RUNG wire#powerrail
      { S7_Templates := "SrcType := DInt" } EQ_Contact(in1 := "Unit1.Em4.ControlNodes".sideTapeLoading.sequence.status.currentStep, in2 := #JOB_2_STEP_50)
      Contact( "Unit1.Em4.ControlNodes".sideTapeLoading.sequence.status.seqActive )
      wire#w1
      I_Contact( "Unit1.Em4.ControlNodes".cmSideTapeCutterClampBwdFwd.monitoring.inWorkPos )
      Coil( "Unit1.Em4.ControlNodes".sideTapeLoading."step".action1[250] )
   END_RUNG
   RUNG wire#w1
      Contact( "Unit1.Em4.ControlNodes".cmSideTapeCutterClampBwdFwd.monitoring.inWorkPos )
      Coil( "Unit1.Em4.ControlNodes".sideTapeLoading."step".transition1[250] )
   END_RUNG
   RUNG wire#w1
      Contact( "Unit1.Em4.ControlNodes".sideTapeLoading."step".transition1[250] )
      { S7_Templates := "time_type := Time" } #statTonTime[250].TON(pt := T#500ms, et =>)
      Move(in := #JOB_2_STEP_60, out1 => "Unit1.Em4.ControlNodes".sideTapeLoading.sequence.status.nextStep)
   END_RUNG
   // the same network as SCL:
   #_w1 := ("Unit1.Em4.ControlNodes".sideTapeLoading.sequence.status.currentStep = #JOB_2_STEP_50) AND "Unit1.Em4.ControlNodes".sideTapeLoading.sequence.status.seqActive;
   "Unit1.Em4.ControlNodes".sideTapeLoading."step".action1[250] := #_w1 AND NOT "Unit1.Em4.ControlNodes".cmSideTapeCutterClampBwdFwd.monitoring.inWorkPos;
   "Unit1.Em4.ControlNodes".sideTapeLoading."step".transition1[250] := #_w1 AND "Unit1.Em4.ControlNodes".cmSideTapeCutterClampBwdFwd.monitoring.inWorkPos;
   #statTonTime[250].TON(IN := #_w1 AND "Unit1.Em4.ControlNodes".sideTapeLoading."step".transition1[250],
                         PT := T#500ms);
   IF #statTonTime[250].Q THEN
       "Unit1.Em4.ControlNodes".sideTapeLoading.sequence.status.nextStep := #JOB_2_STEP_60;
   END_IF;
END_REGION

REGION Network 21: Step[260] : Side Tape Tension Backward
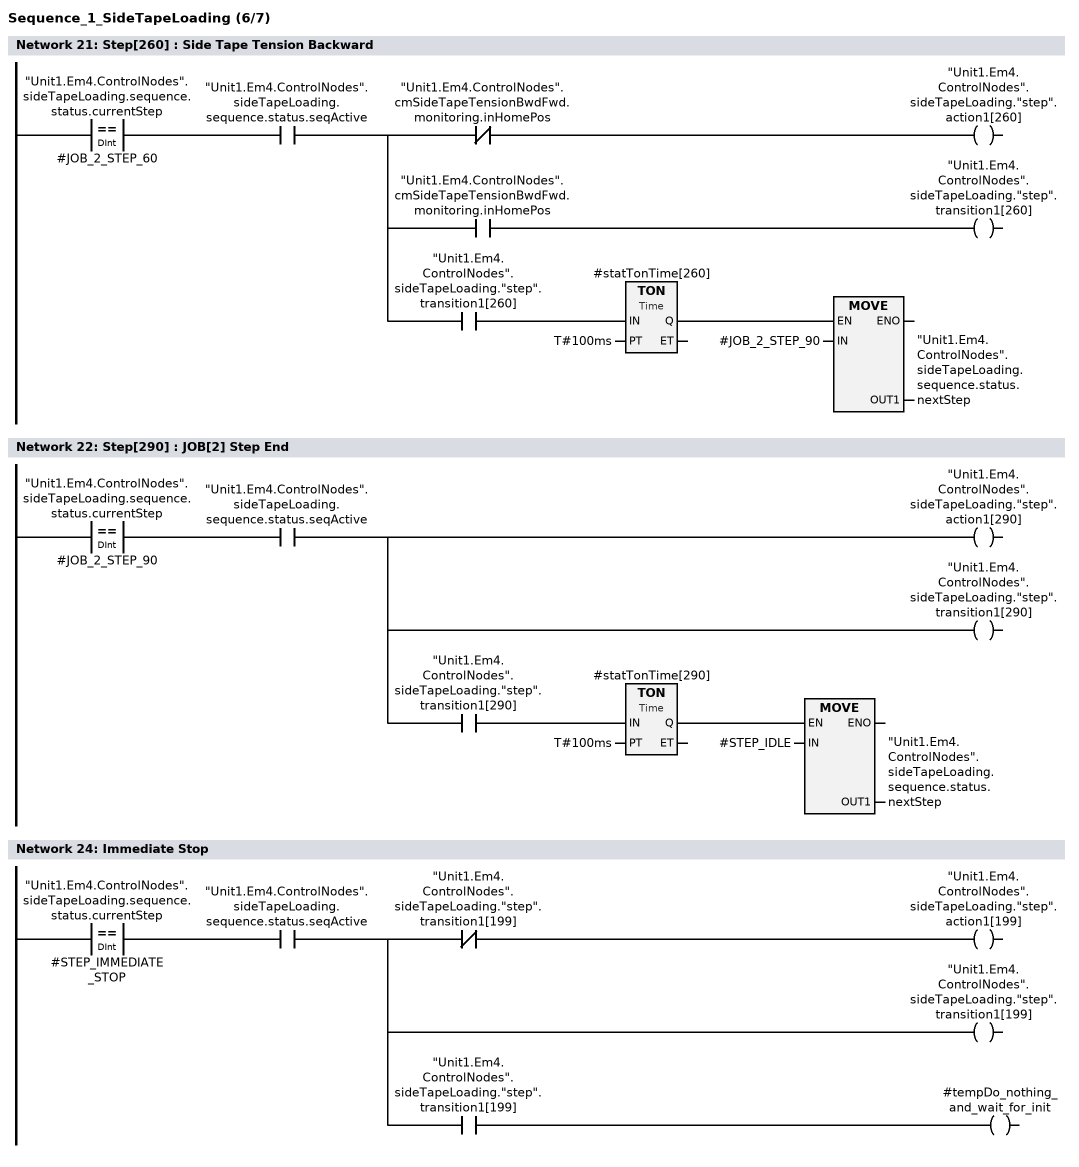
   RUNG wire#powerrail
      { S7_Templates := "SrcType := DInt" } EQ_Contact(in1 := "Unit1.Em4.ControlNodes".sideTapeLoading.sequence.status.currentStep, in2 := #JOB_2_STEP_60)
      Contact( "Unit1.Em4.ControlNodes".sideTapeLoading.sequence.status.seqActive )
      wire#w1
      I_Contact( "Unit1.Em4.ControlNodes".cmSideTapeTensionBwdFwd.monitoring.inHomePos )
      Coil( "Unit1.Em4.ControlNodes".sideTapeLoading."step".action1[260] )
   END_RUNG
   RUNG wire#w1
      Contact( "Unit1.Em4.ControlNodes".cmSideTapeTensionBwdFwd.monitoring.inHomePos )
      Coil( "Unit1.Em4.ControlNodes".sideTapeLoading."step".transition1[260] )
   END_RUNG
   RUNG wire#w1
      Contact( "Unit1.Em4.ControlNodes".sideTapeLoading."step".transition1[260] )
      { S7_Templates := "time_type := Time" } #statTonTime[260].TON(pt := T#100ms, et =>)
      Move(in := #JOB_2_STEP_90, out1 => "Unit1.Em4.ControlNodes".sideTapeLoading.sequence.status.nextStep)
   END_RUNG
   // the same network as SCL:
   #_w1 := ("Unit1.Em4.ControlNodes".sideTapeLoading.sequence.status.currentStep = #JOB_2_STEP_60) AND "Unit1.Em4.ControlNodes".sideTapeLoading.sequence.status.seqActive;
   "Unit1.Em4.ControlNodes".sideTapeLoading."step".action1[260] := #_w1 AND NOT "Unit1.Em4.ControlNodes".cmSideTapeTensionBwdFwd.monitoring.inHomePos;
   "Unit1.Em4.ControlNodes".sideTapeLoading."step".transition1[260] := #_w1 AND "Unit1.Em4.ControlNodes".cmSideTapeTensionBwdFwd.monitoring.inHomePos;
   #statTonTime[260].TON(IN := #_w1 AND "Unit1.Em4.ControlNodes".sideTapeLoading."step".transition1[260],
                         PT := T#100ms);
   IF #statTonTime[260].Q THEN
       "Unit1.Em4.ControlNodes".sideTapeLoading.sequence.status.nextStep := #JOB_2_STEP_90;
   END_IF;
END_REGION

REGION Network 22: Step[290] : JOB[2] Step End
   RUNG wire#powerrail
      { S7_Templates := "SrcType := DInt" } EQ_Contact(in1 := "Unit1.Em4.ControlNodes".sideTapeLoading.sequence.status.currentStep, in2 := #JOB_2_STEP_90)
      Contact( "Unit1.Em4.ControlNodes".sideTapeLoading.sequence.status.seqActive )
      wire#w1
      Coil( "Unit1.Em4.ControlNodes".sideTapeLoading."step".action1[290] )
   END_RUNG
   RUNG wire#w1
      Coil( "Unit1.Em4.ControlNodes".sideTapeLoading."step".transition1[290] )
   END_RUNG
   RUNG wire#w1
      Contact( "Unit1.Em4.ControlNodes".sideTapeLoading."step".transition1[290] )
      { S7_Templates := "time_type := Time" } #statTonTime[290].TON(pt := T#100ms, et =>)
      Move(in := #STEP_IDLE, out1 => "Unit1.Em4.ControlNodes".sideTapeLoading.sequence.status.nextStep)
   END_RUNG
   // the same network as SCL:
   "Unit1.Em4.ControlNodes".sideTapeLoading."step".action1[290] := ("Unit1.Em4.ControlNodes".sideTapeLoading.sequence.status.currentStep = #JOB_2_STEP_90) AND "Unit1.Em4.ControlNodes".sideTapeLoading.sequence.status.seqActive;
   "Unit1.Em4.ControlNodes".sideTapeLoading."step".transition1[290] := ("Unit1.Em4.ControlNodes".sideTapeLoading.sequence.status.currentStep = #JOB_2_STEP_90) AND "Unit1.Em4.ControlNodes".sideTapeLoading.sequence.status.seqActive;
   #statTonTime[290].TON(IN := ("Unit1.Em4.ControlNodes".sideTapeLoading.sequence.status.currentStep = #JOB_2_STEP_90) AND "Unit1.Em4.ControlNodes".sideTapeLoading.sequence.status.seqActive AND "Unit1.Em4.ControlNodes".sideTapeLoading."step".transition1[290],
                         PT := T#100ms);
   IF #statTonTime[290].Q THEN
       "Unit1.Em4.ControlNodes".sideTapeLoading.sequence.status.nextStep := #STEP_IDLE;
   END_IF;
END_REGION

REGION Network 23: *************** IMMEDIATE STOP ****************
END_REGION

REGION Network 24: Immediate Stop
   RUNG wire#powerrail
      { S7_Templates := "SrcType := DInt" } EQ_Contact(in1 := "Unit1.Em4.ControlNodes".sideTapeLoading.sequence.status.currentStep, in2 := #STEP_IMMEDIATE_STOP)
      Contact( "Unit1.Em4.ControlNodes".sideTapeLoading.sequence.status.seqActive )
      wire#w1
      I_Contact( "Unit1.Em4.ControlNodes".sideTapeLoading."step".transition1[199] )
      Coil( "Unit1.Em4.ControlNodes".sideTapeLoading."step".action1[199] )
   END_RUNG
   RUNG wire#w1
      Coil( "Unit1.Em4.ControlNodes".sideTapeLoading."step".transition1[199] )
   END_RUNG
   RUNG wire#w1
      Contact( "Unit1.Em4.ControlNodes".sideTapeLoading."step".transition1[199] )
      Coil( #tempDo_nothing_and_wait_for_init )
   END_RUNG
   // the same network as SCL:
   #_w1 := ("Unit1.Em4.ControlNodes".sideTapeLoading.sequence.status.currentStep = #STEP_IMMEDIATE_STOP) AND "Unit1.Em4.ControlNodes".sideTapeLoading.sequence.status.seqActive;
   "Unit1.Em4.ControlNodes".sideTapeLoading."step".action1[199] := #_w1 AND NOT "Unit1.Em4.ControlNodes".sideTapeLoading."step".transition1[199];
   "Unit1.Em4.ControlNodes".sideTapeLoading."step".transition1[199] := #_w1;
   #tempDo_nothing_and_wait_for_init := #_w1 AND "Unit1.Em4.ControlNodes".sideTapeLoading."step".transition1[199];
END_REGION

REGION Network 25: *************** STATUS **********************
END_REGION

REGION Network 26: Sequence Status
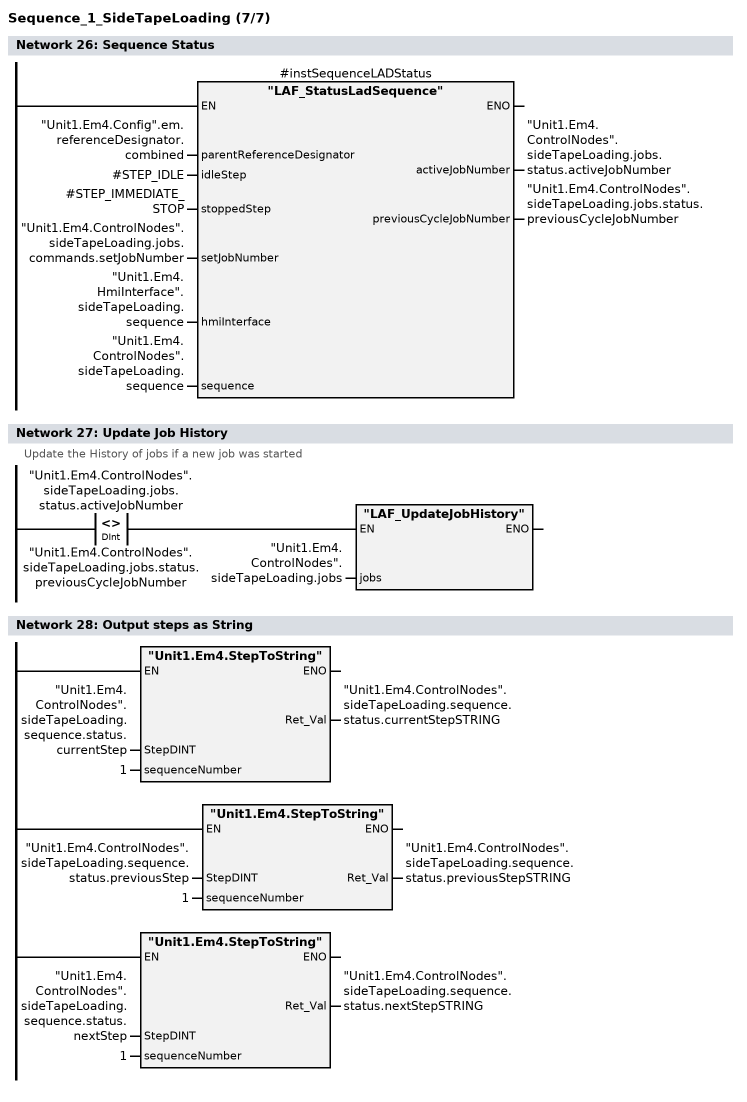
   RUNG wire#powerrail
      #instSequenceLADStatus(parentReferenceDesignator := "Unit1.Em4.Config".em.referenceDesignator.combined, idleStep := #STEP_IDLE, stoppedStep := #STEP_IMMEDIATE_STOP, setJobNumber := "Unit1.Em4.ControlNodes".sideTapeLoading.jobs.commands.setJobNumber, hmiInterface := "Unit1.Em4.HmiInterface".sideTapeLoading.sequence, sequence := "Unit1.Em4.ControlNodes".sideTapeLoading.sequence, activeJobNumber => "Unit1.Em4.ControlNodes".sideTapeLoading.jobs.status.activeJobNumber, previousCycleJobNumber => "Unit1.Em4.ControlNodes".sideTapeLoading.jobs.status.previousCycleJobNumber)
   END_RUNG
   // the same network as SCL:
   #instSequenceLADStatus(parentReferenceDesignator := "Unit1.Em4.Config".em.referenceDesignator.combined,   // "LAF_StatusLadSequence"
                          idleStep := #STEP_IDLE,
                          stoppedStep := #STEP_IMMEDIATE_STOP,
                          setJobNumber := "Unit1.Em4.ControlNodes".sideTapeLoading.jobs.commands.setJobNumber,
                          hmiInterface := "Unit1.Em4.HmiInterface".sideTapeLoading.sequence,
                          sequence := "Unit1.Em4.ControlNodes".sideTapeLoading.sequence,
                          activeJobNumber => "Unit1.Em4.ControlNodes".sideTapeLoading.jobs.status.activeJobNumber,
                          previousCycleJobNumber => "Unit1.Em4.ControlNodes".sideTapeLoading.jobs.status.previousCycleJobNumber);
END_REGION

REGION Network 27: Update Job History
   // Update the History of jobs if a new job was started
   RUNG wire#powerrail
      { S7_Templates := "SrcType := DInt" } NE_Contact(in1 := "Unit1.Em4.ControlNodes".sideTapeLoading.jobs.status.activeJobNumber, in2 := "Unit1.Em4.ControlNodes".sideTapeLoading.jobs.status.previousCycleJobNumber)
      "LAF_UpdateJobHistory"(jobs := "Unit1.Em4.ControlNodes".sideTapeLoading.jobs)
   END_RUNG
   // the same network as SCL:
   IF "Unit1.Em4.ControlNodes".sideTapeLoading.jobs.status.activeJobNumber <> "Unit1.Em4.ControlNodes".sideTapeLoading.jobs.status.previousCycleJobNumber THEN
       "LAF_UpdateJobHistory"(jobs := "Unit1.Em4.ControlNodes".sideTapeLoading.jobs);
   END_IF;
END_REGION

REGION Network 28: Output steps as String
   RUNG wire#powerrail
      "Unit1.Em4.StepToString"(StepDINT := "Unit1.Em4.ControlNodes".sideTapeLoading.sequence.status.currentStep, sequenceNumber := 1, Ret_Val => "Unit1.Em4.ControlNodes".sideTapeLoading.sequence.status.currentStepSTRING)
   END_RUNG
   RUNG wire#powerrail
      "Unit1.Em4.StepToString"(StepDINT := "Unit1.Em4.ControlNodes".sideTapeLoading.sequence.status.previousStep, sequenceNumber := 1, Ret_Val => "Unit1.Em4.ControlNodes".sideTapeLoading.sequence.status.previousStepSTRING)
   END_RUNG
   RUNG wire#powerrail
      "Unit1.Em4.StepToString"(StepDINT := "Unit1.Em4.ControlNodes".sideTapeLoading.sequence.status.nextStep, sequenceNumber := 1, Ret_Val => "Unit1.Em4.ControlNodes".sideTapeLoading.sequence.status.nextStepSTRING)
   END_RUNG
   // the same network as SCL:
   "Unit1.Em4.ControlNodes".sideTapeLoading.sequence.status.currentStepSTRING := "Unit1.Em4.StepToString"(StepDINT := "Unit1.Em4.ControlNodes".sideTapeLoading.sequence.status.currentStep,
                           sequenceNumber := 1);
   "Unit1.Em4.ControlNodes".sideTapeLoading.sequence.status.previousStepSTRING := "Unit1.Em4.StepToString"(StepDINT := "Unit1.Em4.ControlNodes".sideTapeLoading.sequence.status.previousStep,
                           sequenceNumber := 1);
   "Unit1.Em4.ControlNodes".sideTapeLoading.sequence.status.nextStepSTRING := "Unit1.Em4.StepToString"(StepDINT := "Unit1.Em4.ControlNodes".sideTapeLoading.sequence.status.nextStep,
                           sequenceNumber := 1);
END_REGION
END_FUNCTION_BLOCK
